Fanuc KAREL source: kd00003.KL

-- PROVISIONAL review KL for V1013-1; original PC SHA256 bee933cc9a4938a1abdbfe02e32fe2ec66c4898226b773ca46440482df595673
-- Incomplete behavior may be omitted. Consult companion uncertainty JSON. Do not deploy.
PROGRAM KD00003
%NOLOCKGROUP
-- UNRESOLVED_DECL I type=fd0010
-- UNRESOLVED_DECL J type=fd0010
-- UNRESOLVED_DECL B type=fd0012
-- UNRESOLVED_DECL R type=fd0011
-- UNRESOLVED_DECL S type=fd1f50
BEGIN
  -- UNRESOLVED_PC offsets 5-12; opcodes 9D,23
  -- UNRESOLVED_PC offsets 17-21; opcodes 7F
END KD00003
